// Mitsubishi GX Works2 project: CODE   PLC: FX2N/FX2NC

PROGRAM MAIN
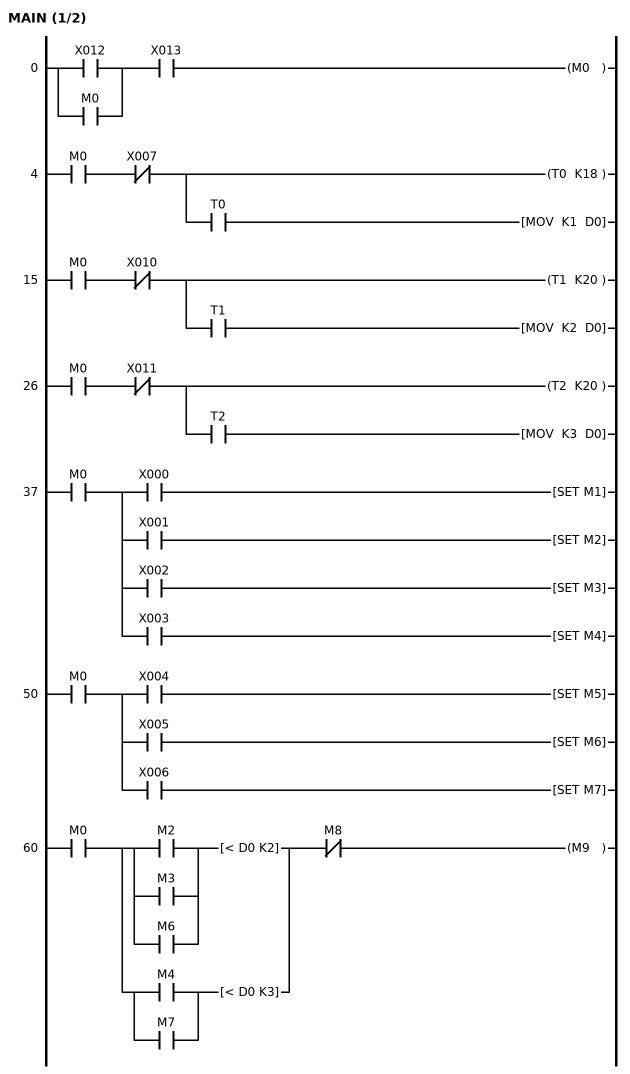
0     LD      X012
      OR      M0
      AND     X013
      OUT     M0
4     LD      M0
      ANI     X007
      OUT     T0 K18
      AND     T0
      MOV     K1 D0
15    LD      M0
      ANI     X010
      OUT     T1 K20
      AND     T1
      MOV     K2 D0
26    LD      M0
      ANI     X011
      OUT     T2 K20
      AND     T2
      MOV     K3 D0
37    LD      M0
      MPS
      AND     X000
      SET     M1
      MRD
      AND     X001
      SET     M2
      MRD
      AND     X002
      SET     M3
      MPP
      AND     X003
      SET     M4
50    LD      M0
      MPS
      AND     X004
      SET     M5
      MRD
      AND     X005
      SET     M6
      MPP
      AND     X006
      SET     M7
60    LD      M0
      LD      M2
      OR      M3
      OR      M6
      AND<    D0 K2
      LD      M4
      OR      M7
      AND<    D0 K3
      ORB
      ANB
      ANI     M8
      OUT     M9
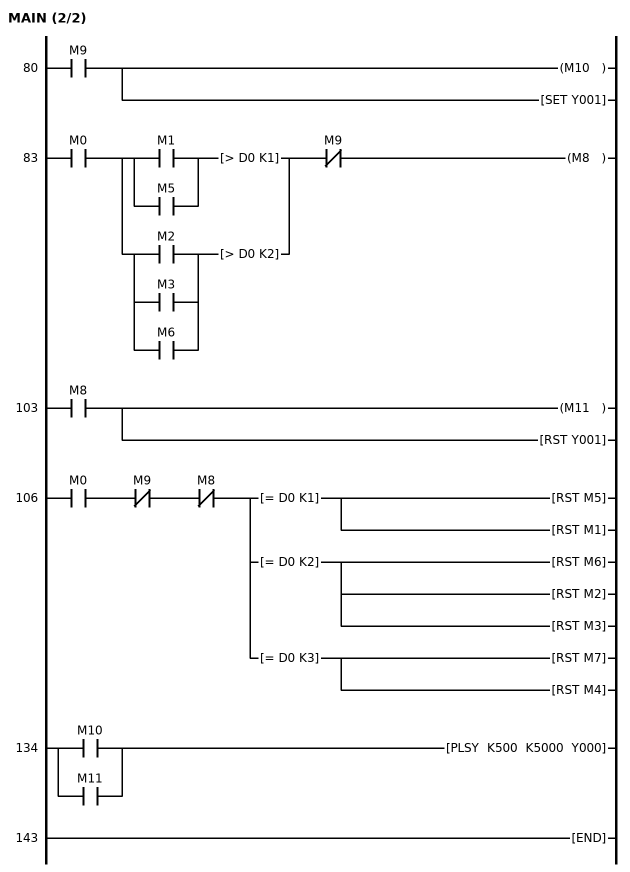
80    LD      M9
      OUT     M10
      SET     Y001
83    LD      M0
      LD      M1
      OR      M5
      AND>    D0 K1
      LD      M2
      OR      M3
      OR      M6
      AND>    D0 K2
      ORB
      ANB
      ANI     M9
      OUT     M8
103   LD      M8
      OUT     M11
      RST     Y001
106   LD      M0
      ANI     M9
      ANI     M8
      MPS
      AND=    D0 K1
      RST     M5
      RST     M1
      MRD
      AND=    D0 K2
      RST     M6
      RST     M2
      RST     M3
      MPP
      AND=    D0 K3
      RST     M7
      RST     M4
134   LD      M10
      OR      M11
      PLSY    K500 K5000 Y000
143   END
END_PROGRAM
